// TIA Portal V17 export
// export: Created 2023-02-13T11:05:53.8511626Z, ExportSetting WithDefaults, DisplayName Totally Integrated Automation Portal, DisplayVersion V17, DisplayName TIA Portal Openness, DisplayVersion V17, DisplayName TIA Portal Teamcenter Gateway, DisplayVersion V17, DisplayName TIA Portal Version Control Interface, DisplayVersion V17, DisplayName SINAMICS Startdrive Advanced, DisplayVersion V17, DisplayName SINAMICS Startdrive G130, G150, S120, S150, SINAMICS MV, S210, DisplayVersion V17, DisplayName SINAMICS Startdrive G110M, G120, G120C, G120D, G120P, G115D, DisplayVersion V17, DisplayName STEP 7 Professional, DisplayVersion V17, DisplayName STEP 7 Safety, DisplayVersion V17, DisplayName WinCC Professional, DisplayVersion V17
VAR_GLOBAL   // PLC tag table "RIO Storage Panel"
   "PS-01 Storage" AT %I54.7 : Bool;   // PRESSURE SWITCH PNEUMATIC VALVE
   "Receive CIP Enable Filling Cryovac" AT %I55.0 : Bool;   // MAIN CIP SUPPLY LINE PRODUCT FROM THE-4 VALVE CLOSE POSITION
   "Receive Product Request Filling Cryovac" AT %I55.1 : Bool;   // MAIN CIP SUPPLY TO STORAGE TANK T-23.00 VALVE CLOSE POSITION
   "Receive CIP Enable Filling ZB" AT %I55.2 : Bool;   // MAIN CIP SUPPLY LINE TO STORAGE TANK T-23.00 VALVE CLOSE POSITION
   "Receive Product Request Filling ZB" AT %I55.3 : Bool;   // MAIN CIP SUPPLY LINE STORAGE TANK T-24.00 VALVE CLOSE POSITION
   "Receive CIP Enable Filling Jonan" AT %I55.4 : Bool;   // MAIN CIP SUPPLY LINE STORAGE TANK T-24.00 VALVE CLOSE POSITION
   "Receive Product Request Filling Jonan" AT %I55.5 : Bool;   // MAIN CIP SUPPLY STORAGE TANK T-25.00 .0
   "Receive CIP Enable Filling FF Winpack" AT %I55.6 : Bool;
   "Receive Product Request Filling FF Winpack" AT %I55.7 : Bool;
   "LT-23.01" AT %IW57 : Int;   // LEVEL TRANSMITTER STORAGE TANK T-23.00
   "LT-24.01" AT %IW59 : Int;   // LEVEL TRANSMITTER STORAGE TANK T-24.00
   "LT-33.01" AT %IW61 : Int;   // LEVEL TRANSMITTER STORAGE TANK T-33.00
   "LT-34.01" AT %IW63 : Int;   // LEVEL TRANSMITTER STORAGE TANK T-34.00
   "LT-35.01" AT %IW65 : Int;   // LEVEL TRANSMITTER STORAGE TANK T-35.00
   "FS-23.01" AT %I53.0 : Bool;   // Flow Switch Transfer Pump P-23.01
   "FS-24.01" AT %I53.1 : Bool;   // Flow Switch Transfer Pump P-24.01
   "FS-34.01" AT %I53.2 : Bool;   // Flow Switch Transfer Pump P-34.01
   "FS-35.01" AT %I53.3 : Bool;   // Flow Switch Transfer Pump P-35.01
   "Receive CIP Enable Filling Jerry Can" AT %I56.0 : Bool;
   "Receive CIP Enable Filling Volpack Pouch" AT %I56.2 : Bool;
   "Receive CIP Enable Filling Mespack New" AT %I56.4 : Bool;
   "Receive CIP Enable Filling Mespack DM" AT %I56.6 : Bool;
   "Receive Product Request Filling Jerry Can" AT %I56.1 : Bool;
   "Receive Product Request Filling Volpack Pouch" AT %I56.3 : Bool;
   "Receive Product Request Filling Mespack New" AT %I56.5 : Bool;
   "Receive Product Request Filling Mespack DM" AT %I56.7 : Bool;
   "Receive CIP Enable Filling Mespack P1" AT %I73.0 : Bool;
   "Receive Product Request Filling Mespack P1" AT %I73.1 : Bool;
   "LT-79.01" AT %IW67 : Int;
   "Potentio Cryovac Pump" AT %IW655 : Int;
   "LT-81.01" AT %IW657 : Int;
   "LT-84.01" AT %IW663 : Int;
   "LT-82.01" AT %IW661 : Int;
   "XA-82.00 Feedback" AT %I54.0 : Bool;   // Feedback Agi ST-16
   "AV-23.01" AT %Q16.0 : Bool;
   "AV-23.02" AT %Q16.1 : Bool;
   "AV-23.03" AT %Q16.2 : Bool;
   "AV-23.04" AT %Q16.3 : Bool;
   "AV-23.05" AT %Q16.4 : Bool;
   "AV-23.06" AT %Q16.5 : Bool;
   "AV-23.07" AT %Q16.6 : Bool;
   "AV-23.08" AT %Q16.7 : Bool;
   "AV-24.01" AT %Q17.0 : Bool;
   "AV-24.02" AT %Q17.1 : Bool;
   "AV-24.03" AT %Q17.2 : Bool;
   "AV-24.04" AT %Q17.3 : Bool;
   "AV-24.05" AT %Q17.4 : Bool;
   "AV-24.06" AT %Q17.5 : Bool;
   "AV-24.13" AT %Q17.6 : Bool;
   "AV-24.14" AT %Q17.7 : Bool;
   "AV-29.01" AT %Q18.0 : Bool;
   "AV-29.02" AT %Q18.1 : Bool;
   "AV-29.03" AT %Q18.2 : Bool;
   "AV-29.04" AT %Q18.3 : Bool;
   "AV-29.06" AT %Q18.4 : Bool;
   "AV-33.01" AT %Q18.5 : Bool;
   "AV-33.02" AT %Q18.6 : Bool;
   "AV-33.03" AT %Q18.7 : Bool;
   "AV-33.04" AT %Q19.0 : Bool;
   "AV-33.05" AT %Q19.1 : Bool;
   "AV-33.06" AT %Q19.2 : Bool;
   "AV-33.07" AT %Q19.3 : Bool;
   "AV-33.08" AT %Q19.4 : Bool;
   "AV-33.09" AT %Q19.5 : Bool;
   "AV-34.09" AT %Q56.0 : Bool;
   "AV-34.10" AT %Q56.1 : Bool;
   "AV-34.11" AT %Q56.2 : Bool;
   "AV-34.12" AT %Q56.3 : Bool;
   "AV-35.01" AT %Q56.4 : Bool;
   "AV-35.02" AT %Q56.5 : Bool;
   "AV-35.03" AT %Q56.6 : Bool;
   "AV-35.04" AT %Q56.7 : Bool;
   "AV-35.05" AT %Q57.0 : Bool;
   "AV-35.06" AT %Q57.1 : Bool;
   "AV-35.07" AT %Q57.2 : Bool;
   "AV-35.08" AT %Q57.3 : Bool;
   "AV-39.01" AT %Q57.4 : Bool;
   "AV-39.02" AT %Q57.5 : Bool;
   "AV-39.03" AT %Q57.6 : Bool;
   "AV-39.04" AT %Q57.7 : Bool;
   "AV-39.06" AT %Q58.0 : Bool;
   "AV-33.10" AT %Q19.6 : Bool;
   "AV-33.11" AT %Q19.7 : Bool;
   "AV-34.01" AT %Q20.0 : Bool;
   "AV-34.02" AT %Q20.1 : Bool;
   "AV-34.03" AT %Q20.2 : Bool;
   "AV-34.04" AT %Q20.3 : Bool;
   "AV-34.05" AT %Q20.4 : Bool;
   "AV-34.06" AT %Q20.5 : Bool;
   "AV-34.07" AT %Q20.6 : Bool;
   "AV-34.08" AT %Q20.7 : Bool;
   "AV-24.15" AT %Q58.1 : Bool;
   "Freq-meter Cryovac Pump Speed" AT %QW60 : Int;
   "AV-24.16" AT %Q58.2 : Bool;
   "AV-79.01" AT %Q58.3 : Bool;
   "AV-79.02" AT %Q82.0 : Bool;
   "AV-79.03" AT %Q82.1 : Bool;
   "AV-79.04" AT %Q82.2 : Bool;
   "AV-79.05" AT %Q82.3 : Bool;
   "AV-79.06" AT %Q82.4 : Bool;
   "AV-79.07" AT %Q82.5 : Bool;
   "AV-79.08" AT %Q82.6 : Bool;
   "AV-79.09" AT %Q82.7 : Bool;
   "AV-79.10" AT %Q83.0 : Bool;
   "AV-79.13" AT %Q83.1 : Bool;
   "AV-79.14" AT %Q83.2 : Bool;
   "AV-79.15" AT %Q83.3 : Bool;
   "AV-79.16" AT %Q83.4 : Bool;
   "AV-79.17" AT %Q83.5 : Bool;
   "AV-81.01" AT %Q83.6 : Bool;
   "AV-81.02" AT %Q83.7 : Bool;
   "AV-81.03" AT %Q84.0 : Bool;
   "AV-81.04" AT %Q84.1 : Bool;
   "AV-81.05" AT %Q84.2 : Bool;
   "AV-81.06" AT %Q84.3 : Bool;
   "AV-81.07" AT %Q84.4 : Bool;
   "AV-81.08" AT %Q84.5 : Bool;
   "AV-81.09" AT %Q84.6 : Bool;
   "AV-81.10" AT %Q84.7 : Bool;
   "AV-81.12" AT %Q85.0 : Bool;
   "AV-81.13" AT %Q85.1 : Bool;
   "AV-81.14" AT %Q85.2 : Bool;
   "AV-85.01" AT %Q85.3 : Bool;
   "AV-85.02" AT %Q85.4 : Bool;
   "AV-85.03" AT %Q85.5 : Bool;
   "AV-85.04" AT %Q85.6 : Bool;
   "AV-85.13" AT %Q85.7 : Bool;
   "AV-85.12" AT %Q86.0 : Bool;
   "AV-85.14" AT %Q86.1 : Bool;
   "AV-85.15" AT %Q86.2 : Bool;
   "AV-85.05" AT %Q86.3 : Bool;
   "AV-85.06" AT %Q86.4 : Bool;
   "AV-85.16" AT %Q86.5 : Bool;
   "AV-85.17" AT %Q86.6 : Bool;
   "AV-85.18" AT %Q86.7 : Bool;
   "AV-85.09" AT %Q87.0 : Bool;
   "AV-85.08" AT %Q87.1 : Bool;
   "AV-85.10" AT %Q87.2 : Bool;
   "AV-85.11" AT %Q87.3 : Bool;
   "AV-84.05" AT %Q87.4 : Bool;
   "AV-84.06" AT %Q87.5 : Bool;
   "AV-84.07" AT %Q87.6 : Bool;
   "AV-84.08" AT %Q87.7 : Bool;
   "AV-84.09" AT %Q88.0 : Bool;
   "AV-84.10" AT %Q88.1 : Bool;
   "AV-84.12" AT %Q88.2 : Bool;
   "AV-84.13" AT %Q88.3 : Bool;
   "AV-84.14" AT %Q88.4 : Bool;
   "XA-82.00 OUT" AT %Q4.0 : Bool;
   spare_ST1 AT %Q4.1 : Bool;
   spare_ST2 AT %Q4.2 : Bool;
   "AV-79.18" AT %Q88.5 : Bool;
   "AV-79.19" AT %Q88.6 : Bool;
   "AV-79.20" AT %Q88.7 : Bool;
   "AV-24.23" AT %Q89.0 : Bool;
   "AV-24.09" AT %Q89.1 : Bool;
   "AV-24.17" AT %Q89.2 : Bool;
   "AV-24.18" AT %Q89.3 : Bool;
   "AV-24.19" AT %Q89.4 : Bool;
   "AV-24.20" AT %Q89.5 : Bool;
   "AV-24.21" AT %Q89.6 : Bool;
   "AV-24.22" AT %Q89.7 : Bool;
END_VAR
